// Mitsubishi GX Works2 project: AI机程序241210   PLC: FX3S

PROGRAM MAIN
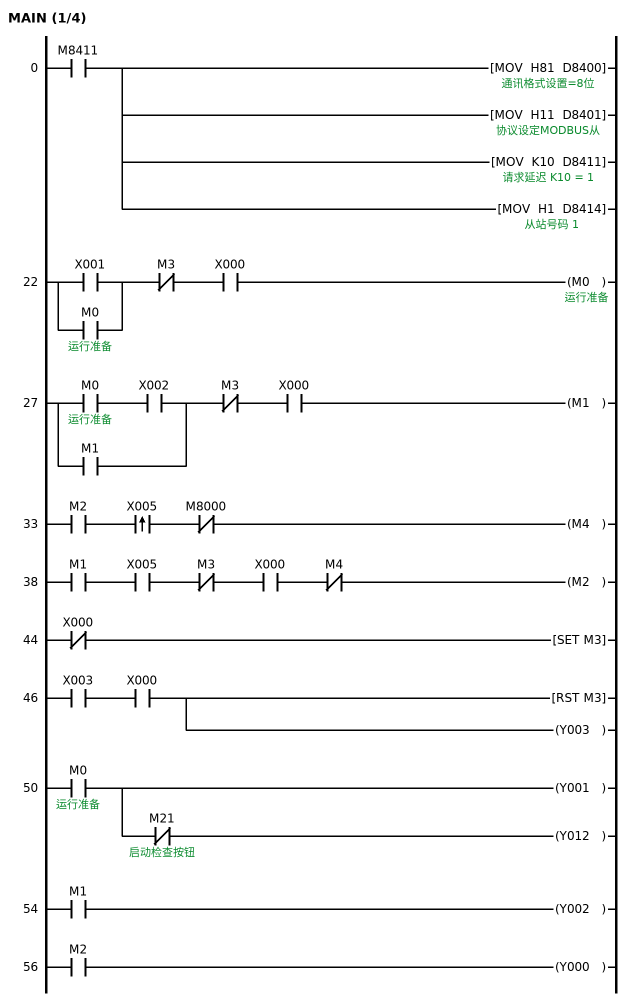
0     LD      M8411
      MOV     H81 D8400  ; 通讯格式设置=8位
      MOV     H11 D8401  ; 协议设定MODBUS从
      MOV     K10 D8411  ; 请求延迟 K10 = 1
      MOV     H1 D8414  ; 从站号码 1
22    LD      X001
      OR      M0  ; 运行准备
      ANI     M3
      AND     X000
      OUT     M0  ; 运行准备
27    LD      M0  ; 运行准备
      AND     X002
      OR      M1
      ANI     M3
      AND     X000
      OUT     M1
33    LD      M2
      ANDP    X005
      ANI     M8000
      OUT     M4
38    LD      M1
      AND     X005
      ANI     M3
      AND     X000
      ANI     M4
      OUT     M2
44    LDI     X000
      SET     M3
46    LD      X003
      AND     X000
      RST     M3
      OUT     Y003
50    LD      M0  ; 运行准备
      OUT     Y001
      ANI     M21  ; 启动检查按钮
      OUT     Y012
54    LD      M1
      OUT     Y002
56    LD      M2
      OUT     Y000
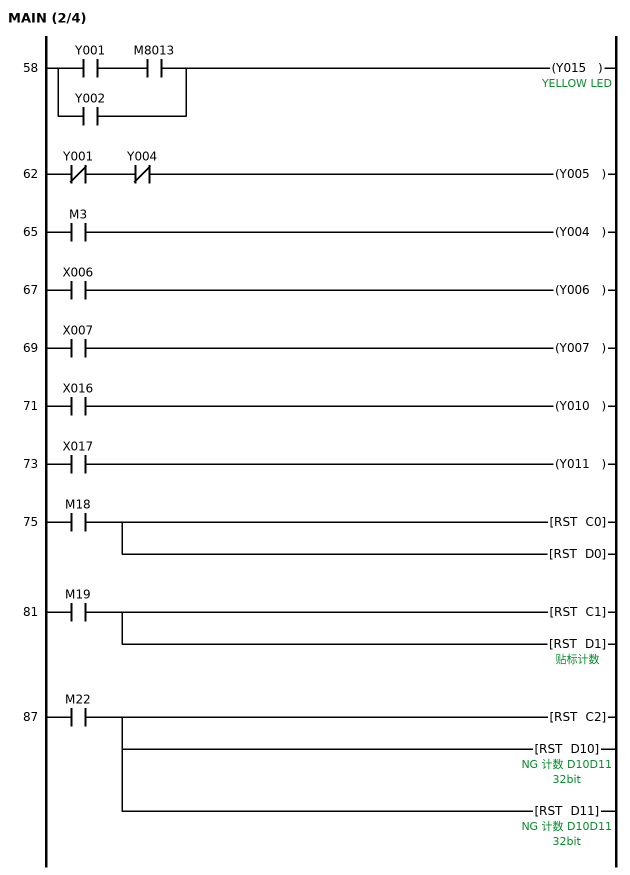
58    LD      Y001
      AND     M8013
      OR      Y002
      OUT     Y015  ; YELLOW LED
62    LDI     Y001
      ANI     Y004
      OUT     Y005
65    LD      M3
      OUT     Y004
67    LD      X006
      OUT     Y006
69    LD      X007
      OUT     Y007
71    LD      X016
      OUT     Y010
73    LD      X017
      OUT     Y011
75    LD      M18
      RST     C0
      RST     D0
81    LD      M19
      RST     C1
      RST     D1  ; 贴标计数
87    LD      M22
      RST     C2
      RST     D10  ; NG 计数 D10D11 32bit
      RST     D11  ; NG 计数 D10D11 32bit
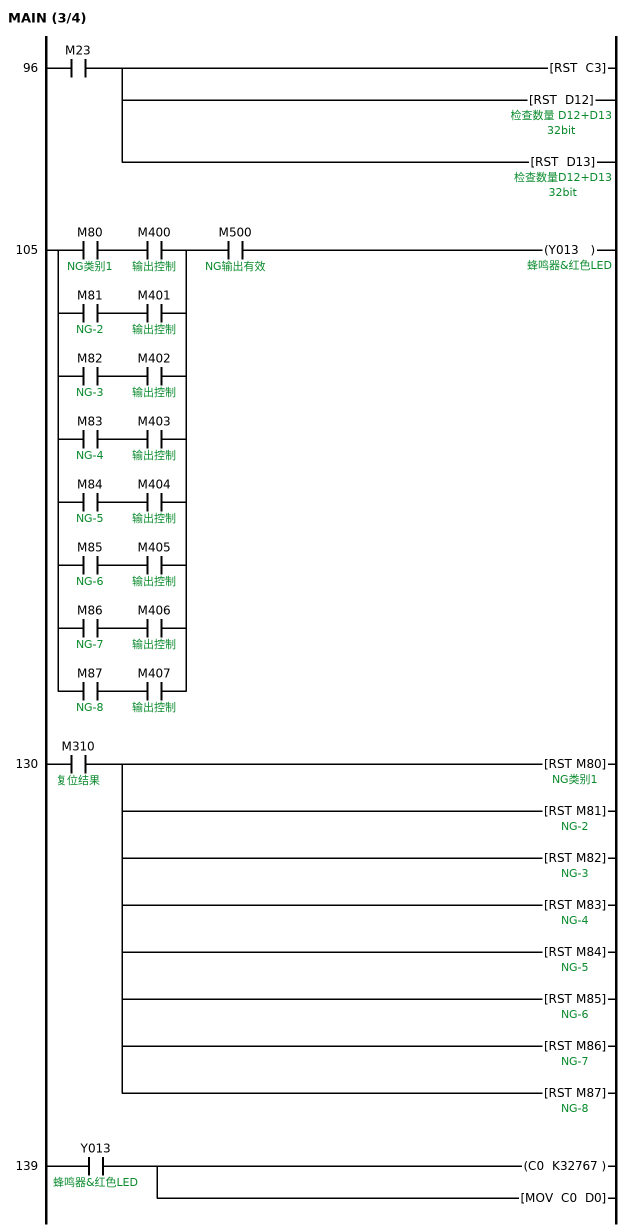
96    LD      M23
      RST     C3
      RST     D12  ; 检查数量 D12+D13 32bit
      RST     D13  ; 检查数量D12+D13 32bit
105   LD      M80  ; NG类别1
      AND     M400  ; 输出控制
      LD      M81  ; NG-2
      AND     M401  ; 输出控制
      ORB
      LD      M82  ; NG-3
      AND     M402  ; 输出控制
      ORB
      LD      M83  ; NG-4
      AND     M403  ; 输出控制
      ORB
      LD      M84  ; NG-5
      AND     M404  ; 输出控制
      ORB
      LD      M85  ; NG-6
      AND     M405  ; 输出控制
      ORB
      LD      M86  ; NG-7
      AND     M406  ; 输出控制
      ORB
      LD      M87  ; NG-8
      AND     M407  ; 输出控制
      ORB
      AND     M500  ; NG输出有效
      OUT     Y013  ; 蜂鸣器&红色LED
130   LD      M310  ; 复位结果
      RST     M80  ; NG类别1
      RST     M81  ; NG-2
      RST     M82  ; NG-3
      RST     M83  ; NG-4
      RST     M84  ; NG-5
      RST     M85  ; NG-6
      RST     M86  ; NG-7
      RST     M87  ; NG-8
139   LD      Y013  ; 蜂鸣器&红色LED
      OUT     C0 K32767
      MOV     C0 D0
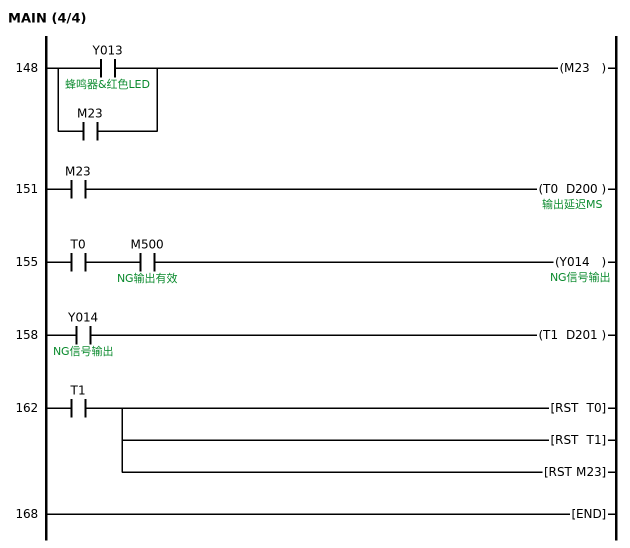
148   LD      Y013  ; 蜂鸣器&红色LED
      OR      M23
      OUT     M23
151   LD      M23
      OUT     T0 D200  ; 输出延迟MS
155   LD      T0
      AND     M500  ; NG输出有效
      OUT     Y014  ; NG信号输出
158   LD      Y014  ; NG信号输出
      OUT     T1 D201
162   LD      T1
      RST     T0
      RST     T1
      RST     M23
168   END
END_PROGRAM

// device comments not shown above
M300  ; 控制开关-GOT
M384  ; 输出控制
M520  ; NG时输出有效
